INTERFACE I_JsonTypeConverter

METHOD PUBLIC DataToJsonString : HRESULT
VAR_INPUT
	Source : I_DataAccess;
	JsonStringAddress : POINTER TO STRING;
	JsonStringSize : UDINT;
END_VAR
END_METHOD

METHOD PUBLIC DataToJsonStringSize : UDINT
VAR_INPUT
	Source : I_DataAccess;
END_VAR
END_METHOD

METHOD PUBLIC JsonStringToData : I_DataDisposer
VAR_INPUT
	JsonStringPointer : POINTER TO STRING;
	Destination : I_DataAccess;
END_VAR
END_METHOD

END_INTERFACE

(* stored: Version 1.1.0.1, ProductVersion 3.1.4024.12
   Itf I_JsonTypeConverter: Id {60a3fa78-0098-0a1a-3ab1-3b6b68cfc3f8}
   Method DataToJsonString: Id {60c6b4b8-8f0a-0677-09c1-c1e681fc871e}
   Method DataToJsonStringSize: Id {80ad02b9-9d7d-0993-2f95-6873be1265b9}
   Method JsonStringToData: Id {c44812b5-9411-003c-1753-de1e9af986e5} *)
